FUNCTION_BLOCK MoldingMachine (* Template for a simple Basic Function Block Type *)
  (* Standard: 61499-2 *)
  (* Version 1.0, 2019-03-27, michael *)
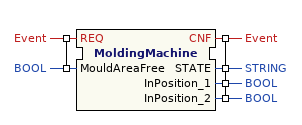
  EVENT_INPUT
    REQ WITH MouldAreaFree; (* Normal Execution Request *)
  END_EVENT
  EVENT_OUTPUT
    CNF WITH STATE, InPosition_1, InPosition_2; (* Execution Confirmation *)
  END_EVENT
  VAR_INPUT
    MouldAreaFree : BOOL := FALSE;
  END_VAR
  VAR_OUTPUT
    STATE : STRING := FALSE; (* Output event qualifier *)
    InPosition_1 : BOOL := FALSE;
    InPosition_2 : BOOL := FALSE;
  END_VAR
  VAR
    LOGIC : BOOL; (* Internal Variable *)
  END_VAR
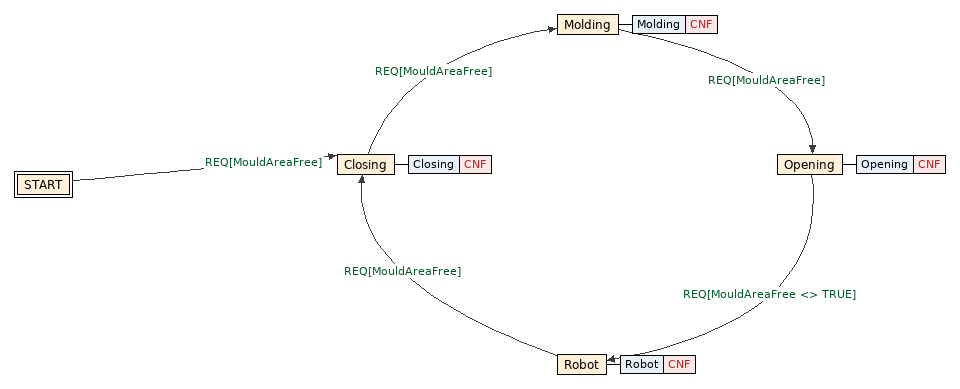
  EC_STATES
    START; (* Initial State *)
    Robot : Robot -> CNF;
    Opening : Opening -> CNF;
    Molding : Molding -> CNF;
    Closing : Closing -> CNF;
  END_STATES
  EC_TRANSITIONS
    Molding TO Opening := REQ[MouldAreaFree];
    Opening TO Robot := REQ[MouldAreaFree <> TRUE];
    Closing TO Molding := REQ[MouldAreaFree];
    START TO Closing := REQ[MouldAreaFree];
    Robot TO Closing := REQ[MouldAreaFree];
  END_TRANSITIONS
  ALGORITHM Molding IN ST: (* new algorithm *)
STATE:="Molding";
InPosition_1:=TRUE;
InPosition_2:=FALSE;
  END_ALGORITHM
  ALGORITHM Opening IN ST: (* new algorithm *)
STATE:="Opening Completed";
InPosition_1:=FALSE;
InPosition_2:=TRUE;
  END_ALGORITHM
  ALGORITHM Robot IN ST: (* new algorithm *)
STATE:="Robot Enters";
InPosition_1:=FALSE;
InPosition_2:=TRUE;
  END_ALGORITHM
  ALGORITHM Closing IN ST: (* new algorithm *)
STATE:="Closing Completed";
InPosition_1:=TRUE;
InPosition_2:=FALSE;
  END_ALGORITHM
END_FUNCTION_BLOCK
